TYPE ST_BaseHMIControlElement_Command :
STRUCT
END_STRUCT
END_TYPE

(* stored: Version 1.1.0.1
   DUT ST_BaseHMIControlElement_Command: Id {432617bd-8195-02f4-0105-2b700bfbf2db} *)
